SUBAPPLICATION Uebung_034 (* Analog-Eingang auf PWM Ausgang *)
  (* Standard: 61499-2 *)
  (* Version 1.0, 2023-10-23, franz *)
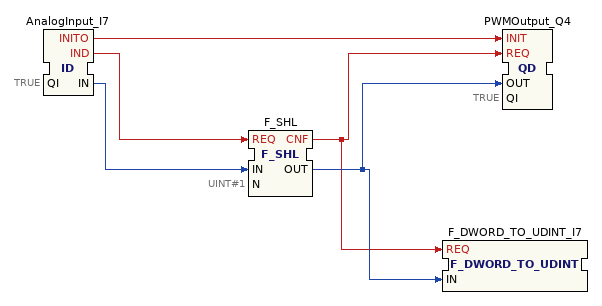
  FBS
    AnalogInput_I7 : ID(QI := TRUE);
    F_DWORD_TO_UDINT_I7 : F_DWORD_TO_UDINT;
    PWMOutput_Q4 : QD(QI := TRUE);
    F_SHL : F_SHL(N := UINT#1);
  END_FBS
  EVENT_CONNECTIONS
    AnalogInput_I7.INITO TO PWMOutput_Q4.INIT;
    AnalogInput_I7.IND TO F_SHL.REQ;
    F_SHL.CNF TO F_DWORD_TO_UDINT_I7.REQ;
    F_SHL.CNF TO PWMOutput_Q4.REQ;
  END_CONNECTIONS
  DATA_CONNECTIONS
    AnalogInput_I7.IN TO F_SHL.IN;
    F_SHL.OUT TO PWMOutput_Q4.OUT;
    F_SHL.OUT TO F_DWORD_TO_UDINT_I7.IN;
  END_CONNECTIONS
END_SUBAPPLICATION
